DATA_BLOCK "dbArchiveParBoiler"
{ S7_Optimized_Access := 'TRUE' }
VERSION : 0.8
"fbArchiveParBoiler"

BEGIN

END_DATA_BLOCK

